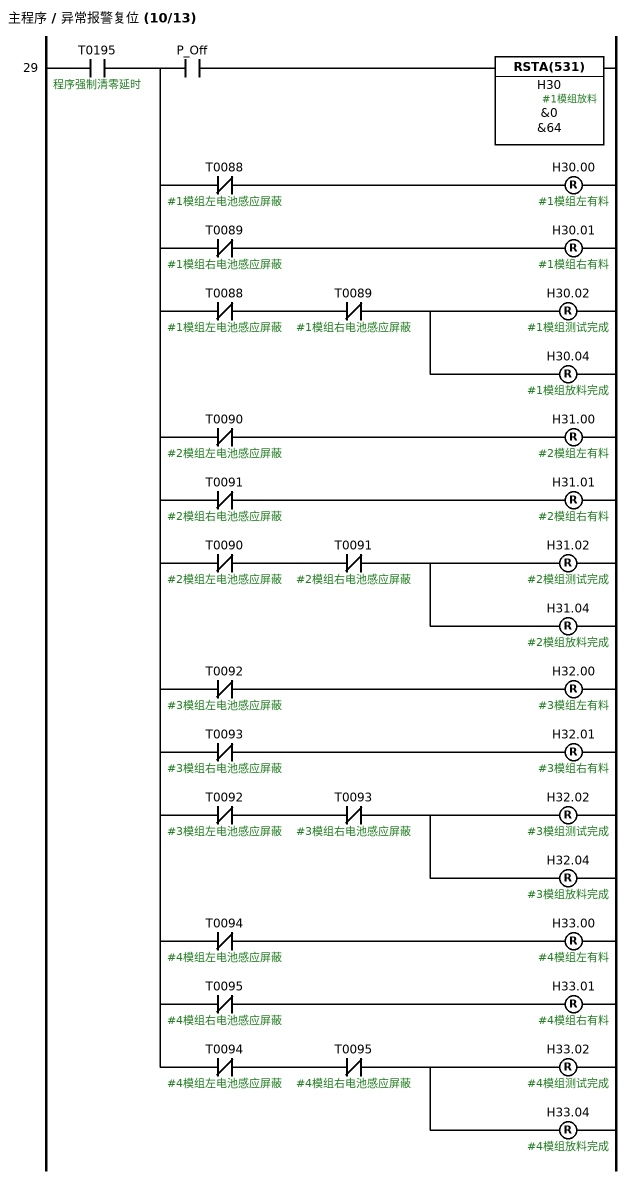
; [picture p17: 主程序 / 异常报警复位, rungs 29-29]
; rung 29
LD T0195  ; 程序强制清零延时
OUT TR0
AND P_Off
RSTA(531) H30 &0 &64  ; #1模组放料
LD TR0
ANDNOT T0088  ; #1模组左电池感应屏蔽
RSET H30.00  ; #1模组左有料
LD TR0
ANDNOT T0089  ; #1模组右电池感应屏蔽
RSET H30.01  ; #1模组右有料
LD TR0
ANDNOT T0088  ; #1模组左电池感应屏蔽
ANDNOT T0089  ; #1模组右电池感应屏蔽
RSET H30.02  ; #1模组测试完成
RSET H30.04  ; #1模组放料完成
LD TR0
ANDNOT T0090  ; #2模组左电池感应屏蔽
RSET H31.00  ; #2模组左有料
LD TR0
ANDNOT T0091  ; #2模组右电池感应屏蔽
RSET H31.01  ; #2模组右有料
LD TR0
ANDNOT T0090  ; #2模组左电池感应屏蔽
ANDNOT T0091  ; #2模组右电池感应屏蔽
RSET H31.02  ; #2模组测试完成
RSET H31.04  ; #2模组放料完成
LD TR0
ANDNOT T0092  ; #3模组左电池感应屏蔽
RSET H32.00  ; #3模组左有料
LD TR0
ANDNOT T0093  ; #3模组右电池感应屏蔽
RSET H32.01  ; #3模组右有料
LD TR0
ANDNOT T0092  ; #3模组左电池感应屏蔽
ANDNOT T0093  ; #3模组右电池感应屏蔽
RSET H32.02  ; #3模组测试完成
RSET H32.04  ; #3模组放料完成
LD TR0
ANDNOT T0094  ; #4模组左电池感应屏蔽
RSET H33.00  ; #4模组左有料
LD TR0
ANDNOT T0095  ; #4模组右电池感应屏蔽
RSET H33.01  ; #4模组右有料
LD TR0
ANDNOT T0094  ; #4模组左电池感应屏蔽
ANDNOT T0095  ; #4模组右电池感应屏蔽
RSET H33.02  ; #4模组测试完成
RSET H33.04  ; #4模组放料完成

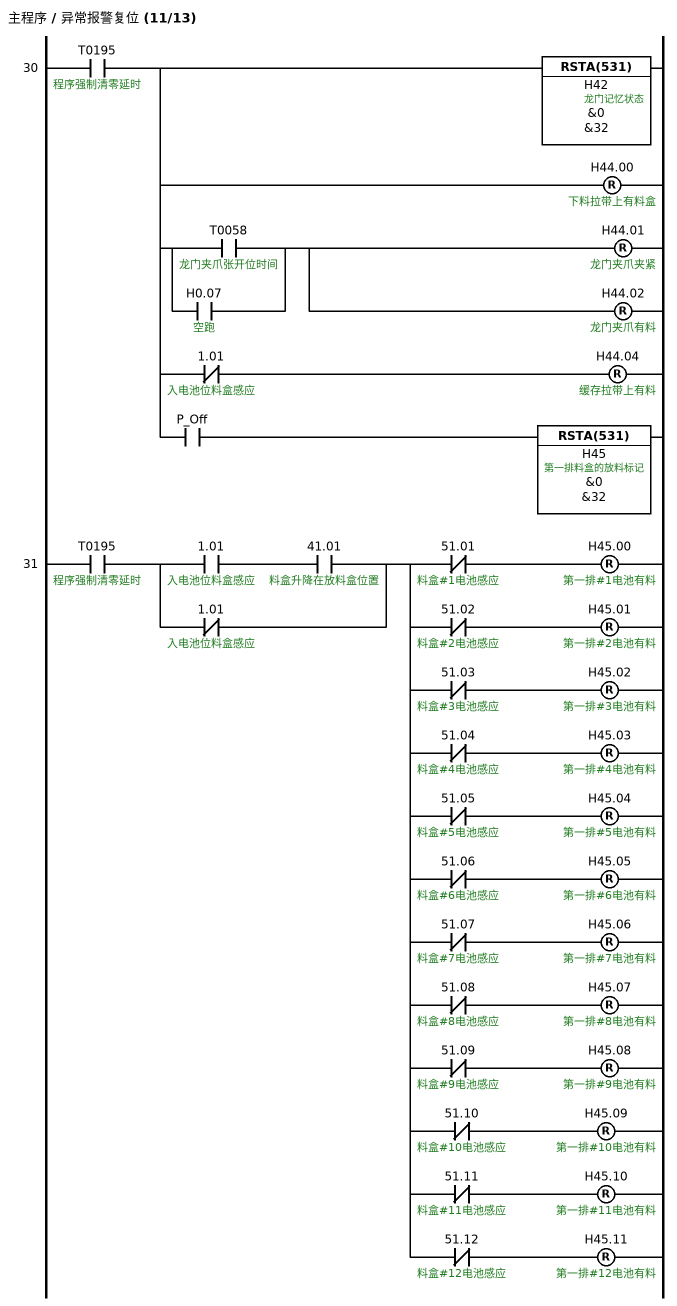
; rung 30
LD T0195  ; 程序强制清零延时
OUT TR0
RSTA(531) H42 &0 &32  ; 龙门记忆状态
RSET H44.00  ; 下料拉带上有料盒
LD T0058  ; 龙门夹爪张开位时间
OR H0.07  ; 空跑
ANDLD
RSET H44.01  ; 龙门夹爪夹紧
RSET H44.02  ; 龙门夹爪有料
LD TR0
ANDNOT 1.01  ; 入电池位料盒感应
RSET H44.04  ; 缓存拉带上有料
LD TR0
AND P_Off
RSTA(531) H45 &0 &32  ; 第一排料盒的放料标记
; rung 31
LD T0195  ; 程序强制清零延时
LD 1.01  ; 入电池位料盒感应
AND 41.01  ; 料盒升降在放料盒位置
ORNOT 1.01  ; 入电池位料盒感应
ANDLD
OUT TR0
ANDNOT 51.01  ; 料盒#1电池感应
RSET H45.00  ; 第一排#1电池有料
LD TR0
ANDNOT 51.02  ; 料盒#2电池感应
RSET H45.01  ; 第一排#2电池有料
LD TR0
ANDNOT 51.03  ; 料盒#3电池感应
RSET H45.02  ; 第一排#3电池有料
LD TR0
ANDNOT 51.04  ; 料盒#4电池感应
RSET H45.03  ; 第一排#4电池有料
LD TR0
ANDNOT 51.05  ; 料盒#5电池感应
RSET H45.04  ; 第一排#5电池有料
LD TR0
ANDNOT 51.06  ; 料盒#6电池感应
RSET H45.05  ; 第一排#6电池有料
LD TR0
ANDNOT 51.07  ; 料盒#7电池感应
RSET H45.06  ; 第一排#7电池有料
LD TR0
ANDNOT 51.08  ; 料盒#8电池感应
RSET H45.07  ; 第一排#8电池有料
LD TR0
ANDNOT 51.09  ; 料盒#9电池感应
RSET H45.08  ; 第一排#9电池有料
LD TR0
ANDNOT 51.10  ; 料盒#10电池感应
RSET H45.09  ; 第一排#10电池有料
LD TR0
ANDNOT 51.11  ; 料盒#11电池感应
RSET H45.10  ; 第一排#11电池有料
LD TR0
ANDNOT 51.12  ; 料盒#12电池感应
RSET H45.11  ; 第一排#12电池有料

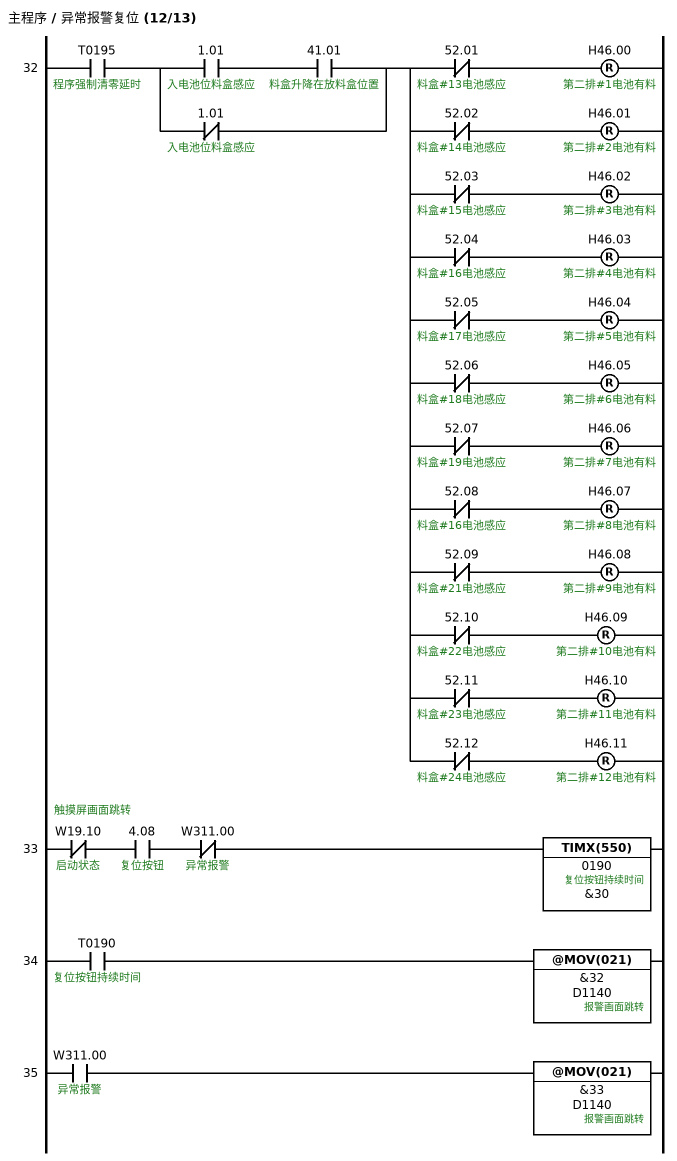
; rung 32
LD T0195  ; 程序强制清零延时
LD 1.01  ; 入电池位料盒感应
AND 41.01  ; 料盒升降在放料盒位置
ORNOT 1.01  ; 入电池位料盒感应
ANDLD
OUT TR0
ANDNOT 52.01  ; 料盒#13电池感应
RSET H46.00  ; 第二排#1电池有料
LD TR0
ANDNOT 52.02  ; 料盒#14电池感应
RSET H46.01  ; 第二排#2电池有料
LD TR0
ANDNOT 52.03  ; 料盒#15电池感应
RSET H46.02  ; 第二排#3电池有料
LD TR0
ANDNOT 52.04  ; 料盒#16电池感应
RSET H46.03  ; 第二排#4电池有料
LD TR0
ANDNOT 52.05  ; 料盒#17电池感应
RSET H46.04  ; 第二排#5电池有料
LD TR0
ANDNOT 52.06  ; 料盒#18电池感应
RSET H46.05  ; 第二排#6电池有料
LD TR0
ANDNOT 52.07  ; 料盒#19电池感应
RSET H46.06  ; 第二排#7电池有料
LD TR0
ANDNOT 52.08  ; 料盒#16电池感应
RSET H46.07  ; 第二排#8电池有料
LD TR0
ANDNOT 52.09  ; 料盒#21电池感应
RSET H46.08  ; 第二排#9电池有料
LD TR0
ANDNOT 52.10  ; 料盒#22电池感应
RSET H46.09  ; 第二排#10电池有料
LD TR0
ANDNOT 52.11  ; 料盒#23电池感应
RSET H46.10  ; 第二排#11电池有料
LD TR0
ANDNOT 52.12  ; 料盒#24电池感应
RSET H46.11  ; 第二排#12电池有料
; rung 33: 触摸屏画面跳转
LDNOT W19.10  ; 启动状态
AND 4.08  ; 复位按钮
ANDNOT W311.00  ; 异常报警
TIMX(550) 0190 &30  ; 复位按钮持续时间
; rung 34
LD T0190  ; 复位按钮持续时间
@MOV(021) &32 D1140  ; 报警画面跳转
; rung 35
LD W311.00  ; 异常报警
@MOV(021) &33 D1140  ; 报警画面跳转

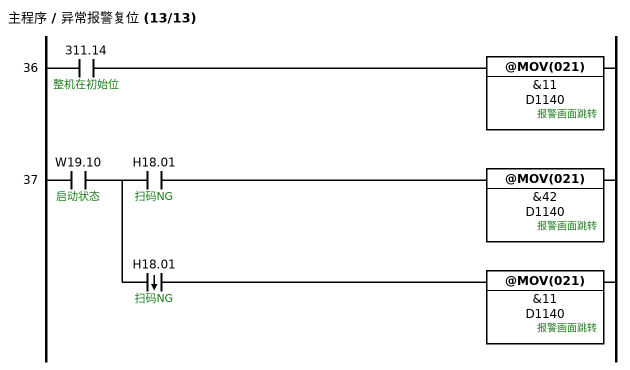
; rung 36
LD 311.14  ; 整机在初始位
@MOV(021) &11 D1140  ; 报警画面跳转
; rung 37
LD W19.10  ; 启动状态
OUT TR0
AND H18.01  ; 扫码NG
@MOV(021) &42 D1140  ; 报警画面跳转
LD TR0
%AND H18.01  ; 扫码NG
@MOV(021) &11 D1140  ; 报警画面跳转

### Section END
; rung 0
END(001)

## Program 传感器 (cyclic task 1)

### Section 感应器屏蔽

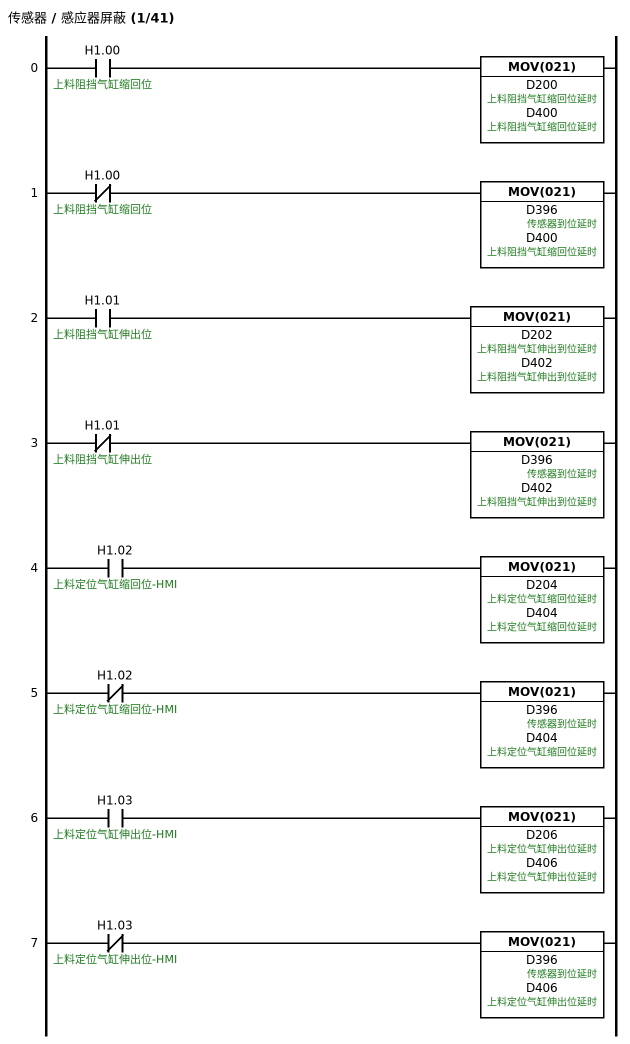
; rung 0
LD H1.00  ; 上料阻挡气缸缩回位
MOV(021) D200 D400  ; 上料阻挡气缸缩回位延时
; rung 1
LDNOT H1.00  ; 上料阻挡气缸缩回位
MOV(021) D396 D400  ; 传感器到位延时, 上料阻挡气缸缩回位延时
; rung 2
LD H1.01  ; 上料阻挡气缸伸出位
MOV(021) D202 D402  ; 上料阻挡气缸伸出到位延时
; rung 3
LDNOT H1.01  ; 上料阻挡气缸伸出位
MOV(021) D396 D402  ; 传感器到位延时, 上料阻挡气缸伸出到位延时
; rung 4
LD H1.02  ; 上料定位气缸缩回位-HMI
MOV(021) D204 D404  ; 上料定位气缸缩回位延时
; rung 5
LDNOT H1.02  ; 上料定位气缸缩回位-HMI
MOV(021) D396 D404  ; 传感器到位延时, 上料定位气缸缩回位延时
; rung 6
LD H1.03  ; 上料定位气缸伸出位-HMI
MOV(021) D206 D406  ; 上料定位气缸伸出位延时
; rung 7
LDNOT H1.03  ; 上料定位气缸伸出位-HMI
MOV(021) D396 D406  ; 传感器到位延时, 上料定位气缸伸出位延时

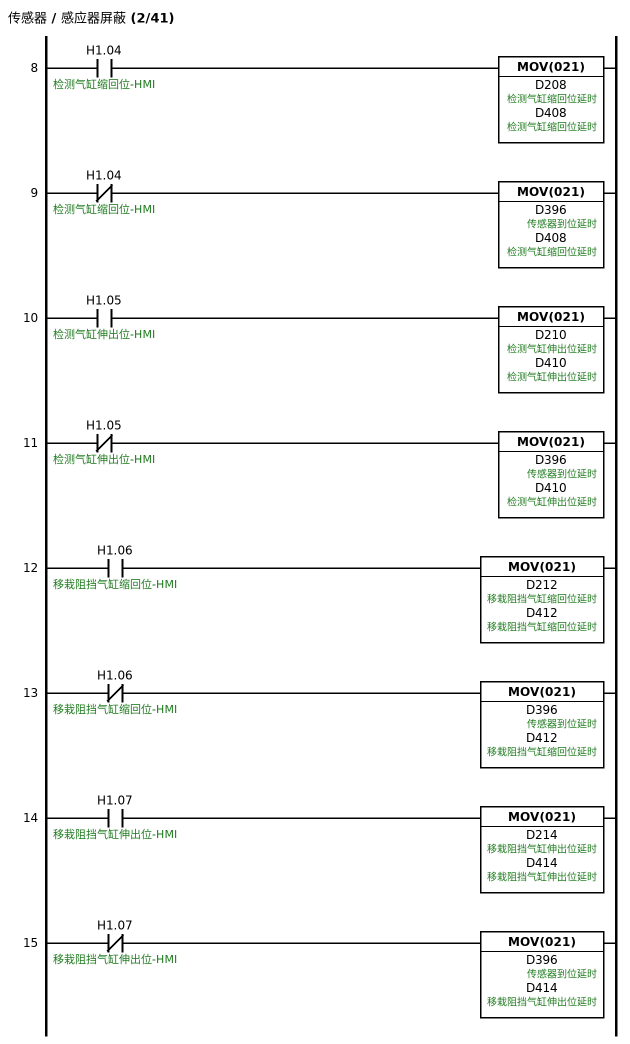
; rung 8
LD H1.04  ; 检测气缸缩回位-HMI
MOV(021) D208 D408  ; 检测气缸缩回位延时
; rung 9
LDNOT H1.04  ; 检测气缸缩回位-HMI
MOV(021) D396 D408  ; 传感器到位延时, 检测气缸缩回位延时
; rung 10
LD H1.05  ; 检测气缸伸出位-HMI
MOV(021) D210 D410  ; 检测气缸伸出位延时
; rung 11
LDNOT H1.05  ; 检测气缸伸出位-HMI
MOV(021) D396 D410  ; 传感器到位延时, 检测气缸伸出位延时
; rung 12
LD H1.06  ; 移栽阻挡气缸缩回位-HMI
MOV(021) D212 D412  ; 移栽阻挡气缸缩回位延时
; rung 13
LDNOT H1.06  ; 移栽阻挡气缸缩回位-HMI
MOV(021) D396 D412  ; 传感器到位延时, 移栽阻挡气缸缩回位延时
; rung 14
LD H1.07  ; 移栽阻挡气缸伸出位-HMI
MOV(021) D214 D414  ; 移栽阻挡气缸伸出位延时
; rung 15
LDNOT H1.07  ; 移栽阻挡气缸伸出位-HMI
MOV(021) D396 D414  ; 传感器到位延时, 移栽阻挡气缸伸出位延时

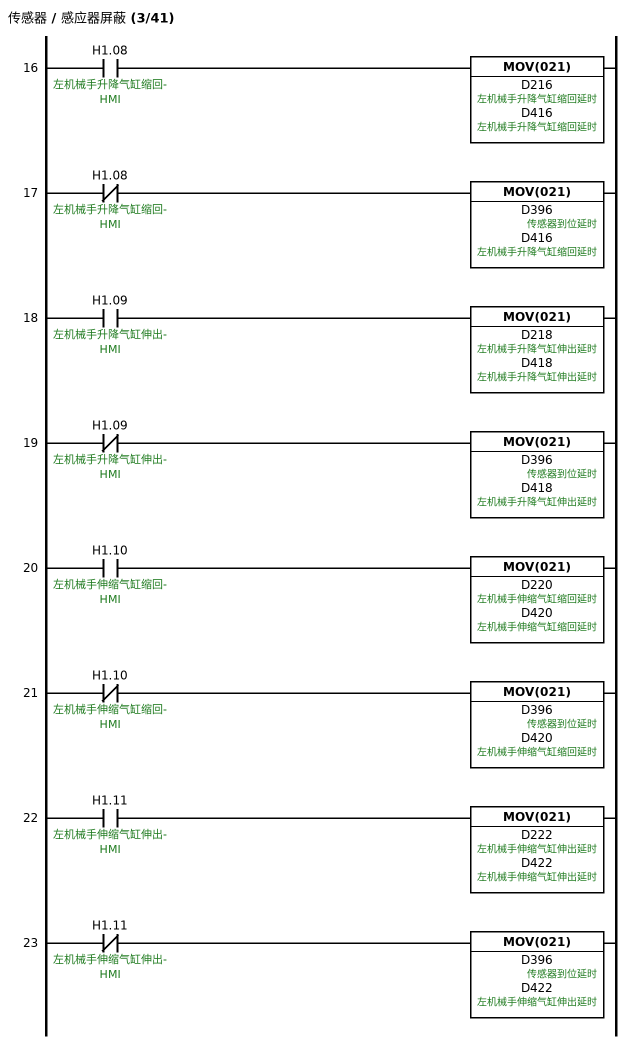
; rung 16
LD H1.08  ; 左机械手升降气缸缩回-HMI
MOV(021) D216 D416  ; 左机械手升降气缸缩回延时
; rung 17
LDNOT H1.08  ; 左机械手升降气缸缩回-HMI
MOV(021) D396 D416  ; 传感器到位延时, 左机械手升降气缸缩回延时
; rung 18
LD H1.09  ; 左机械手升降气缸伸出-HMI
MOV(021) D218 D418  ; 左机械手升降气缸伸出延时
; rung 19
LDNOT H1.09  ; 左机械手升降气缸伸出-HMI
MOV(021) D396 D418  ; 传感器到位延时, 左机械手升降气缸伸出延时
; rung 20
LD H1.10  ; 左机械手伸缩气缸缩回-HMI
MOV(021) D220 D420  ; 左机械手伸缩气缸缩回延时
; rung 21
LDNOT H1.10  ; 左机械手伸缩气缸缩回-HMI
MOV(021) D396 D420  ; 传感器到位延时, 左机械手伸缩气缸缩回延时
; rung 22
LD H1.11  ; 左机械手伸缩气缸伸出-HMI
MOV(021) D222 D422  ; 左机械手伸缩气缸伸出延时
; rung 23
LDNOT H1.11  ; 左机械手伸缩气缸伸出-HMI
MOV(021) D396 D422  ; 传感器到位延时, 左机械手伸缩气缸伸出延时

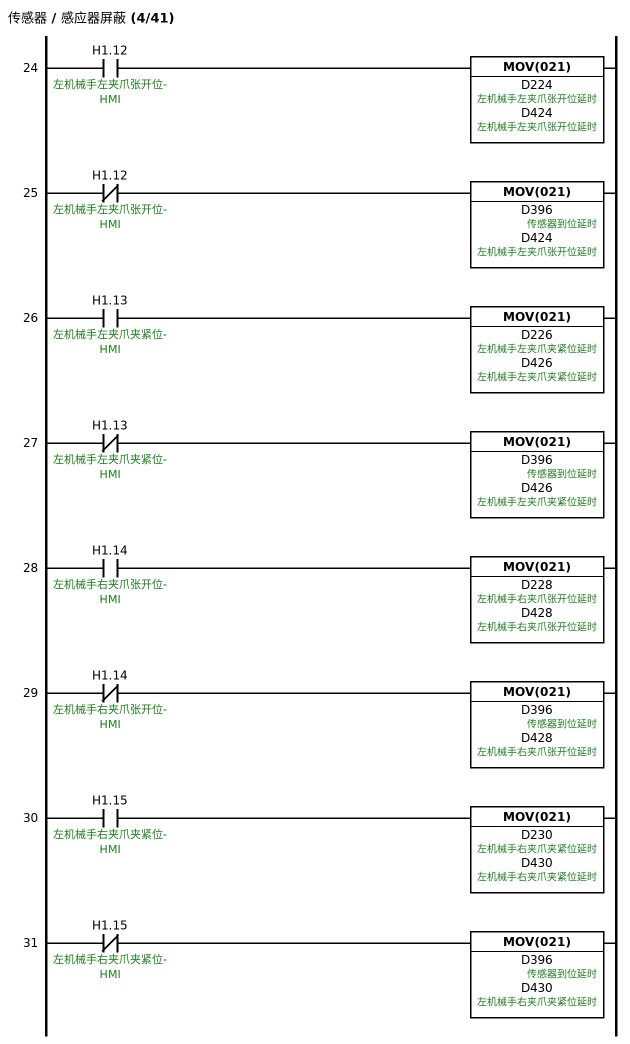
; rung 24
LD H1.12  ; 左机械手左夹爪张开位-HMI
MOV(021) D224 D424  ; 左机械手左夹爪张开位延时
; rung 25
LDNOT H1.12  ; 左机械手左夹爪张开位-HMI
MOV(021) D396 D424  ; 传感器到位延时, 左机械手左夹爪张开位延时
; rung 26
LD H1.13  ; 左机械手左夹爪夹紧位-HMI
MOV(021) D226 D426  ; 左机械手左夹爪夹紧位延时
; rung 27
LDNOT H1.13  ; 左机械手左夹爪夹紧位-HMI
MOV(021) D396 D426  ; 传感器到位延时, 左机械手左夹爪夹紧位延时
; rung 28
LD H1.14  ; 左机械手右夹爪张开位-HMI
MOV(021) D228 D428  ; 左机械手右夹爪张开位延时
; rung 29
LDNOT H1.14  ; 左机械手右夹爪张开位-HMI
MOV(021) D396 D428  ; 传感器到位延时, 左机械手右夹爪张开位延时
; rung 30
LD H1.15  ; 左机械手右夹爪夹紧位-HMI
MOV(021) D230 D430  ; 左机械手右夹爪夹紧位延时
; rung 31
LDNOT H1.15  ; 左机械手右夹爪夹紧位-HMI
MOV(021) D396 D430  ; 传感器到位延时, 左机械手右夹爪夹紧位延时

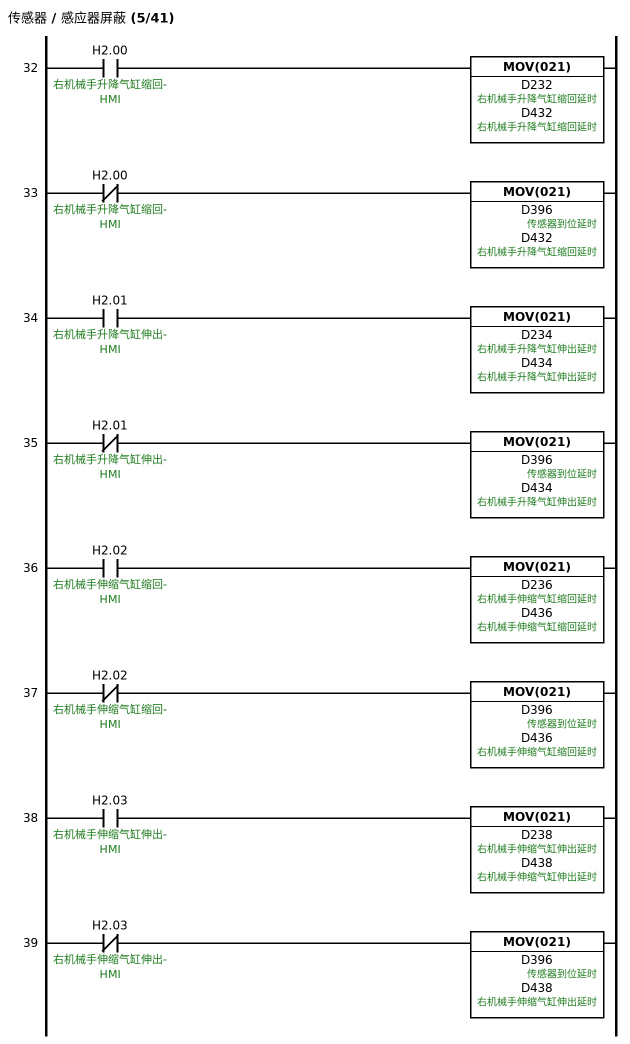
; rung 32
LD H2.00  ; 右机械手升降气缸缩回-HMI
MOV(021) D232 D432  ; 右机械手升降气缸缩回延时
; rung 33
LDNOT H2.00  ; 右机械手升降气缸缩回-HMI
MOV(021) D396 D432  ; 传感器到位延时, 右机械手升降气缸缩回延时
; rung 34
LD H2.01  ; 右机械手升降气缸伸出-HMI
MOV(021) D234 D434  ; 右机械手升降气缸伸出延时
; rung 35
LDNOT H2.01  ; 右机械手升降气缸伸出-HMI
MOV(021) D396 D434  ; 传感器到位延时, 右机械手升降气缸伸出延时
; rung 36
LD H2.02  ; 右机械手伸缩气缸缩回-HMI
MOV(021) D236 D436  ; 右机械手伸缩气缸缩回延时
; rung 37
LDNOT H2.02  ; 右机械手伸缩气缸缩回-HMI
MOV(021) D396 D436  ; 传感器到位延时, 右机械手伸缩气缸缩回延时
; rung 38
LD H2.03  ; 右机械手伸缩气缸伸出-HMI
MOV(021) D238 D438  ; 右机械手伸缩气缸伸出延时
; rung 39
LDNOT H2.03  ; 右机械手伸缩气缸伸出-HMI
MOV(021) D396 D438  ; 传感器到位延时, 右机械手伸缩气缸伸出延时

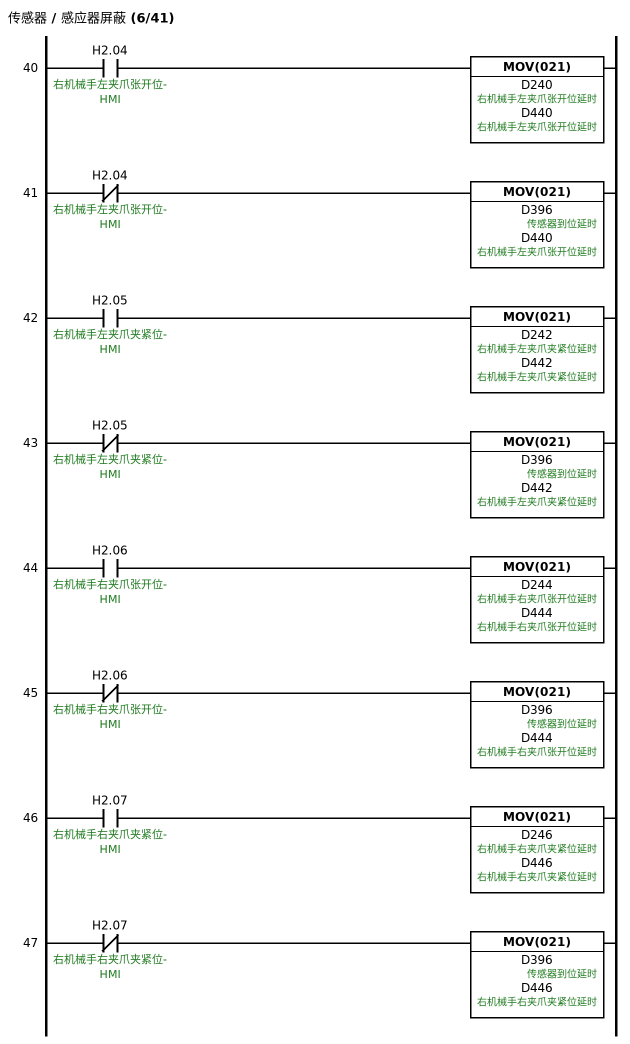
; rung 40
LD H2.04  ; 右机械手左夹爪张开位-HMI
MOV(021) D240 D440  ; 右机械手左夹爪张开位延时
; rung 41
LDNOT H2.04  ; 右机械手左夹爪张开位-HMI
MOV(021) D396 D440  ; 传感器到位延时, 右机械手左夹爪张开位延时
; rung 42
LD H2.05  ; 右机械手左夹爪夹紧位-HMI
MOV(021) D242 D442  ; 右机械手左夹爪夹紧位延时
; rung 43
LDNOT H2.05  ; 右机械手左夹爪夹紧位-HMI
MOV(021) D396 D442  ; 传感器到位延时, 右机械手左夹爪夹紧位延时
; rung 44
LD H2.06  ; 右机械手右夹爪张开位-HMI
MOV(021) D244 D444  ; 右机械手右夹爪张开位延时
; rung 45
LDNOT H2.06  ; 右机械手右夹爪张开位-HMI
MOV(021) D396 D444  ; 传感器到位延时, 右机械手右夹爪张开位延时
; rung 46
LD H2.07  ; 右机械手右夹爪夹紧位-HMI
MOV(021) D246 D446  ; 右机械手右夹爪夹紧位延时
; rung 47
LDNOT H2.07  ; 右机械手右夹爪夹紧位-HMI
MOV(021) D396 D446  ; 传感器到位延时, 右机械手右夹爪夹紧位延时

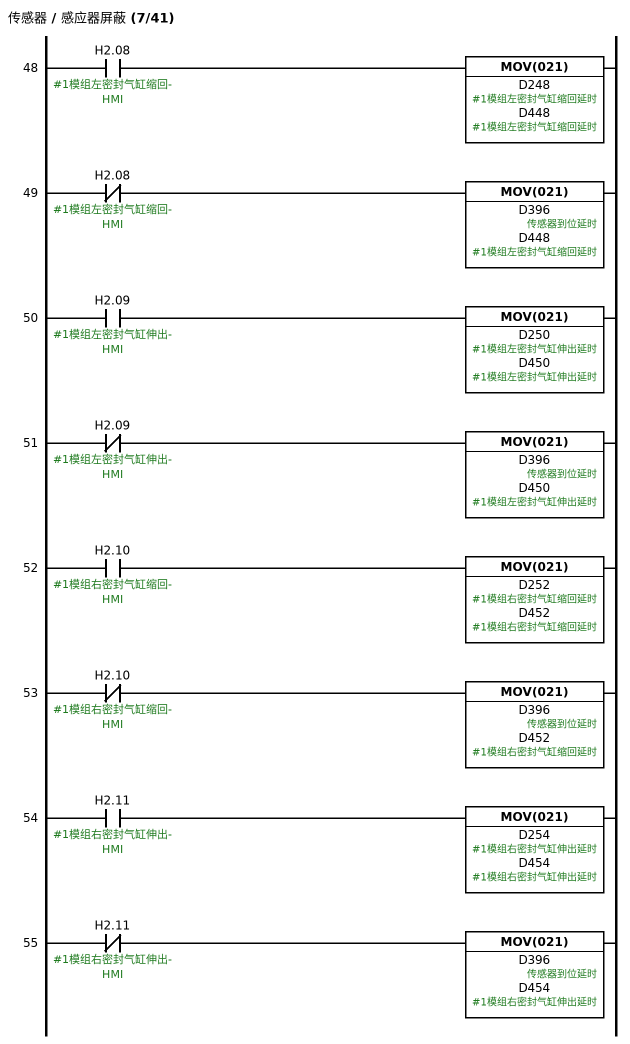
; rung 48
LD H2.08  ; #1模组左密封气缸缩回-HMI
MOV(021) D248 D448  ; #1模组左密封气缸缩回延时
; rung 49
LDNOT H2.08  ; #1模组左密封气缸缩回-HMI
MOV(021) D396 D448  ; 传感器到位延时, #1模组左密封气缸缩回延时
; rung 50
LD H2.09  ; #1模组左密封气缸伸出-HMI
MOV(021) D250 D450  ; #1模组左密封气缸伸出延时
; rung 51
LDNOT H2.09  ; #1模组左密封气缸伸出-HMI
MOV(021) D396 D450  ; 传感器到位延时, #1模组左密封气缸伸出延时
; rung 52
LD H2.10  ; #1模组右密封气缸缩回-HMI
MOV(021) D252 D452  ; #1模组右密封气缸缩回延时
; rung 53
LDNOT H2.10  ; #1模组右密封气缸缩回-HMI
MOV(021) D396 D452  ; 传感器到位延时, #1模组右密封气缸缩回延时
; rung 54
LD H2.11  ; #1模组右密封气缸伸出-HMI
MOV(021) D254 D454  ; #1模组右密封气缸伸出延时
; rung 55
LDNOT H2.11  ; #1模组右密封气缸伸出-HMI
MOV(021) D396 D454  ; 传感器到位延时, #1模组右密封气缸伸出延时

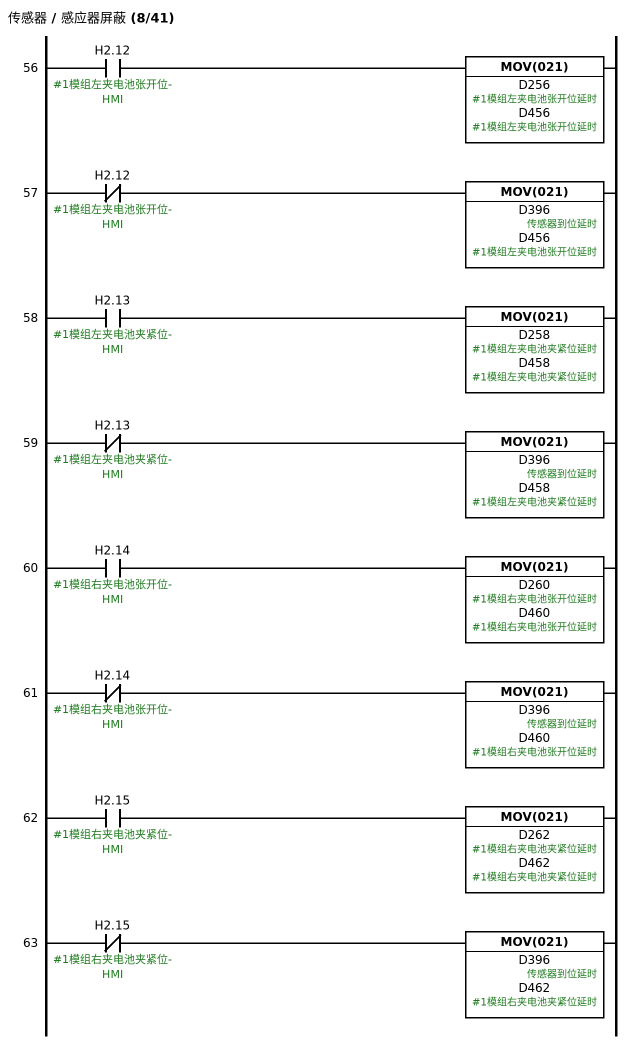
; rung 56
LD H2.12  ; #1模组左夹电池张开位-HMI
MOV(021) D256 D456  ; #1模组左夹电池张开位延时
; rung 57
LDNOT H2.12  ; #1模组左夹电池张开位-HMI
MOV(021) D396 D456  ; 传感器到位延时, #1模组左夹电池张开位延时
; rung 58
LD H2.13  ; #1模组左夹电池夹紧位-HMI
MOV(021) D258 D458  ; #1模组左夹电池夹紧位延时
; rung 59
LDNOT H2.13  ; #1模组左夹电池夹紧位-HMI
MOV(021) D396 D458  ; 传感器到位延时, #1模组左夹电池夹紧位延时
; rung 60
LD H2.14  ; #1模组右夹电池张开位-HMI
MOV(021) D260 D460  ; #1模组右夹电池张开位延时
; rung 61
LDNOT H2.14  ; #1模组右夹电池张开位-HMI
MOV(021) D396 D460  ; 传感器到位延时, #1模组右夹电池张开位延时
; rung 62
LD H2.15  ; #1模组右夹电池夹紧位-HMI
MOV(021) D262 D462  ; #1模组右夹电池夹紧位延时
; rung 63
LDNOT H2.15  ; #1模组右夹电池夹紧位-HMI
MOV(021) D396 D462  ; 传感器到位延时, #1模组右夹电池夹紧位延时

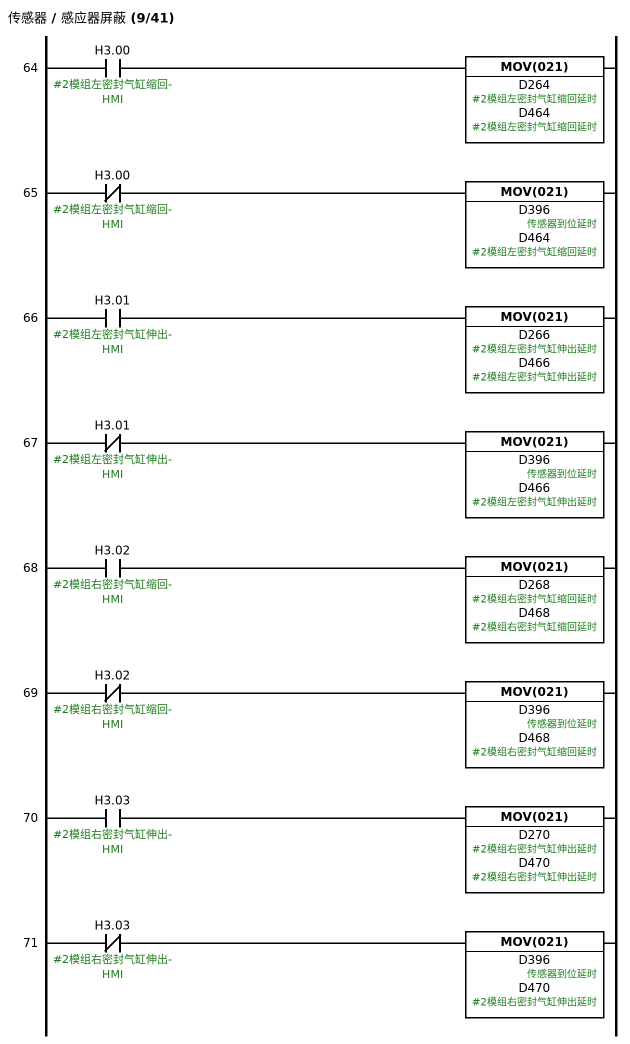
; rung 64
LD H3.00  ; #2模组左密封气缸缩回-HMI
MOV(021) D264 D464  ; #2模组左密封气缸缩回延时
; rung 65
LDNOT H3.00  ; #2模组左密封气缸缩回-HMI
MOV(021) D396 D464  ; 传感器到位延时, #2模组左密封气缸缩回延时
; rung 66
LD H3.01  ; #2模组左密封气缸伸出-HMI
MOV(021) D266 D466  ; #2模组左密封气缸伸出延时
; rung 67
LDNOT H3.01  ; #2模组左密封气缸伸出-HMI
MOV(021) D396 D466  ; 传感器到位延时, #2模组左密封气缸伸出延时
; rung 68
LD H3.02  ; #2模组右密封气缸缩回-HMI
MOV(021) D268 D468  ; #2模组右密封气缸缩回延时
; rung 69
LDNOT H3.02  ; #2模组右密封气缸缩回-HMI
MOV(021) D396 D468  ; 传感器到位延时, #2模组右密封气缸缩回延时
; rung 70
LD H3.03  ; #2模组右密封气缸伸出-HMI
MOV(021) D270 D470  ; #2模组右密封气缸伸出延时
; rung 71
LDNOT H3.03  ; #2模组右密封气缸伸出-HMI
MOV(021) D396 D470  ; 传感器到位延时, #2模组右密封气缸伸出延时

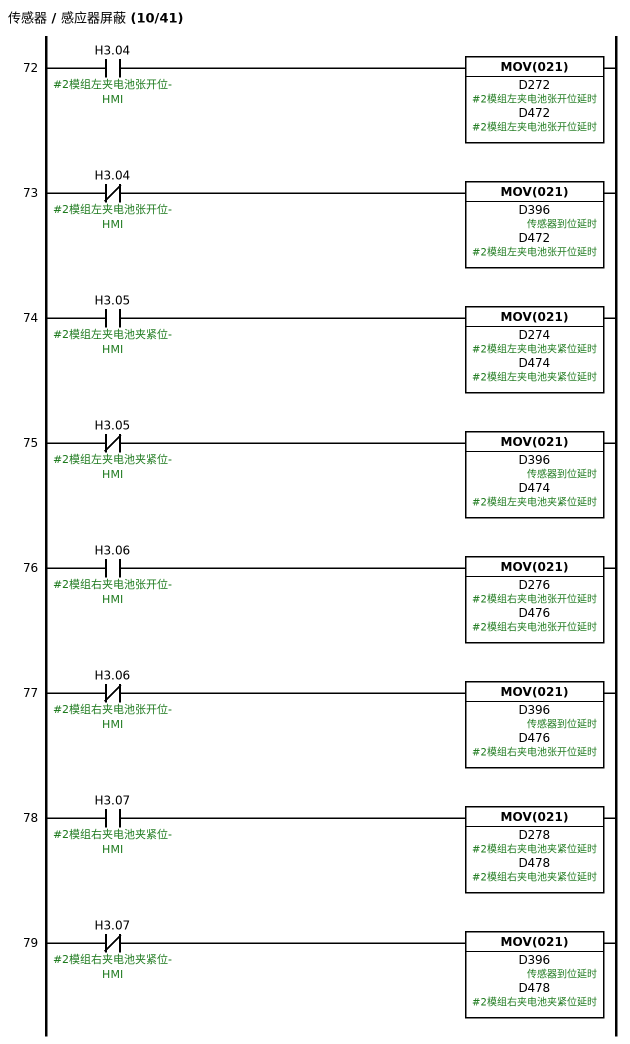
; rung 72
LD H3.04  ; #2模组左夹电池张开位-HMI
MOV(021) D272 D472  ; #2模组左夹电池张开位延时
; rung 73
LDNOT H3.04  ; #2模组左夹电池张开位-HMI
MOV(021) D396 D472  ; 传感器到位延时, #2模组左夹电池张开位延时
; rung 74
LD H3.05  ; #2模组左夹电池夹紧位-HMI
MOV(021) D274 D474  ; #2模组左夹电池夹紧位延时
; rung 75
LDNOT H3.05  ; #2模组左夹电池夹紧位-HMI
MOV(021) D396 D474  ; 传感器到位延时, #2模组左夹电池夹紧位延时
; rung 76
LD H3.06  ; #2模组右夹电池张开位-HMI
MOV(021) D276 D476  ; #2模组右夹电池张开位延时
; rung 77
LDNOT H3.06  ; #2模组右夹电池张开位-HMI
MOV(021) D396 D476  ; 传感器到位延时, #2模组右夹电池张开位延时
; rung 78
LD H3.07  ; #2模组右夹电池夹紧位-HMI
MOV(021) D278 D478  ; #2模组右夹电池夹紧位延时
; rung 79
LDNOT H3.07  ; #2模组右夹电池夹紧位-HMI
MOV(021) D396 D478  ; 传感器到位延时, #2模组右夹电池夹紧位延时

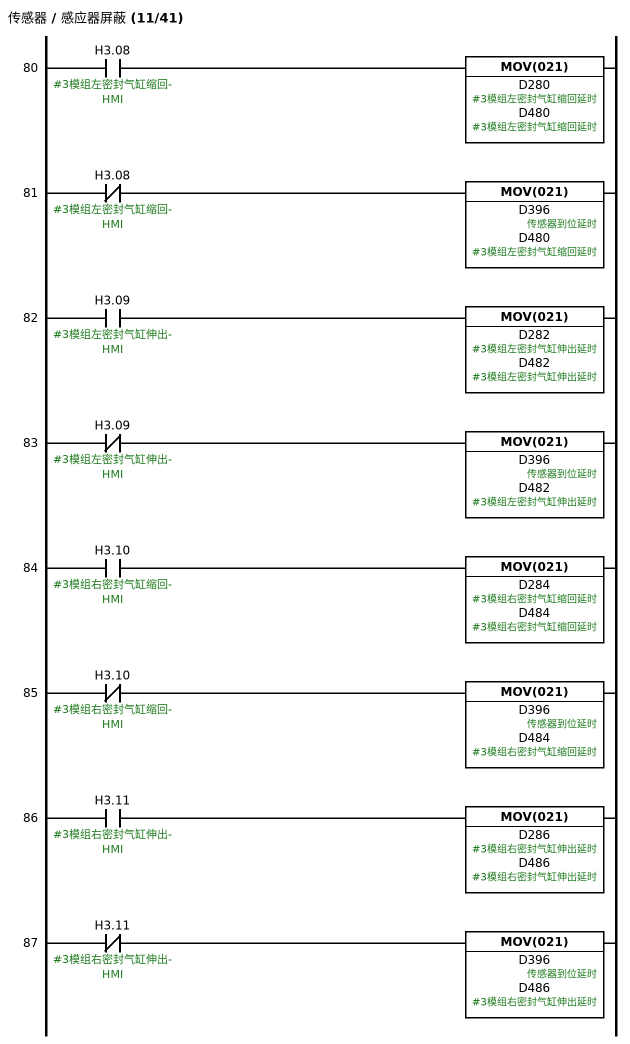
; rung 80
LD H3.08  ; #3模组左密封气缸缩回-HMI
MOV(021) D280 D480  ; #3模组左密封气缸缩回延时
; rung 81
LDNOT H3.08  ; #3模组左密封气缸缩回-HMI
MOV(021) D396 D480  ; 传感器到位延时, #3模组左密封气缸缩回延时
; rung 82
LD H3.09  ; #3模组左密封气缸伸出-HMI
MOV(021) D282 D482  ; #3模组左密封气缸伸出延时
; rung 83
LDNOT H3.09  ; #3模组左密封气缸伸出-HMI
MOV(021) D396 D482  ; 传感器到位延时, #3模组左密封气缸伸出延时
; rung 84
LD H3.10  ; #3模组右密封气缸缩回-HMI
MOV(021) D284 D484  ; #3模组右密封气缸缩回延时
; rung 85
LDNOT H3.10  ; #3模组右密封气缸缩回-HMI
MOV(021) D396 D484  ; 传感器到位延时, #3模组右密封气缸缩回延时
; rung 86
LD H3.11  ; #3模组右密封气缸伸出-HMI
MOV(021) D286 D486  ; #3模组右密封气缸伸出延时
; rung 87
LDNOT H3.11  ; #3模组右密封气缸伸出-HMI
MOV(021) D396 D486  ; 传感器到位延时, #3模组右密封气缸伸出延时

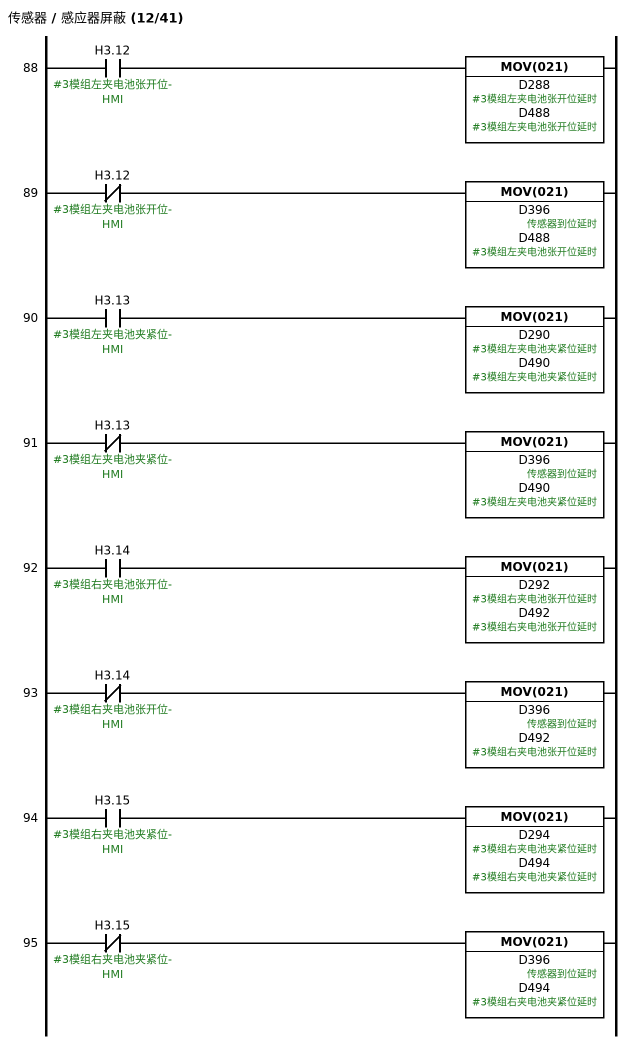
; rung 88
LD H3.12  ; #3模组左夹电池张开位-HMI
MOV(021) D288 D488  ; #3模组左夹电池张开位延时
; rung 89
LDNOT H3.12  ; #3模组左夹电池张开位-HMI
MOV(021) D396 D488  ; 传感器到位延时, #3模组左夹电池张开位延时
; rung 90
LD H3.13  ; #3模组左夹电池夹紧位-HMI
MOV(021) D290 D490  ; #3模组左夹电池夹紧位延时
; rung 91
LDNOT H3.13  ; #3模组左夹电池夹紧位-HMI
MOV(021) D396 D490  ; 传感器到位延时, #3模组左夹电池夹紧位延时
; rung 92
LD H3.14  ; #3模组右夹电池张开位-HMI
MOV(021) D292 D492  ; #3模组右夹电池张开位延时
; rung 93
LDNOT H3.14  ; #3模组右夹电池张开位-HMI
MOV(021) D396 D492  ; 传感器到位延时, #3模组右夹电池张开位延时
; rung 94
LD H3.15  ; #3模组右夹电池夹紧位-HMI
MOV(021) D294 D494  ; #3模组右夹电池夹紧位延时
; rung 95
LDNOT H3.15  ; #3模组右夹电池夹紧位-HMI
MOV(021) D396 D494  ; 传感器到位延时, #3模组右夹电池夹紧位延时

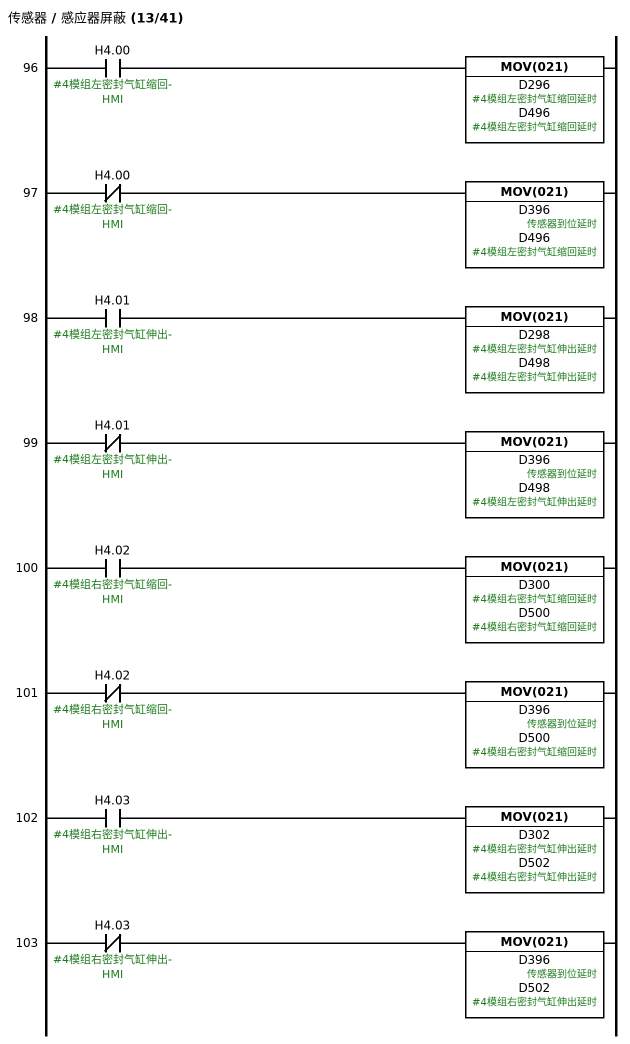
; rung 96
LD H4.00  ; #4模组左密封气缸缩回-HMI
MOV(021) D296 D496  ; #4模组左密封气缸缩回延时
; rung 97
LDNOT H4.00  ; #4模组左密封气缸缩回-HMI
MOV(021) D396 D496  ; 传感器到位延时, #4模组左密封气缸缩回延时
; rung 98
LD H4.01  ; #4模组左密封气缸伸出-HMI
MOV(021) D298 D498  ; #4模组左密封气缸伸出延时
; rung 99
LDNOT H4.01  ; #4模组左密封气缸伸出-HMI
MOV(021) D396 D498  ; 传感器到位延时, #4模组左密封气缸伸出延时
; rung 100
LD H4.02  ; #4模组右密封气缸缩回-HMI
MOV(021) D300 D500  ; #4模组右密封气缸缩回延时
; rung 101
LDNOT H4.02  ; #4模组右密封气缸缩回-HMI
MOV(021) D396 D500  ; 传感器到位延时, #4模组右密封气缸缩回延时
; rung 102
LD H4.03  ; #4模组右密封气缸伸出-HMI
MOV(021) D302 D502  ; #4模组右密封气缸伸出延时
; rung 103
LDNOT H4.03  ; #4模组右密封气缸伸出-HMI
MOV(021) D396 D502  ; 传感器到位延时, #4模组右密封气缸伸出延时

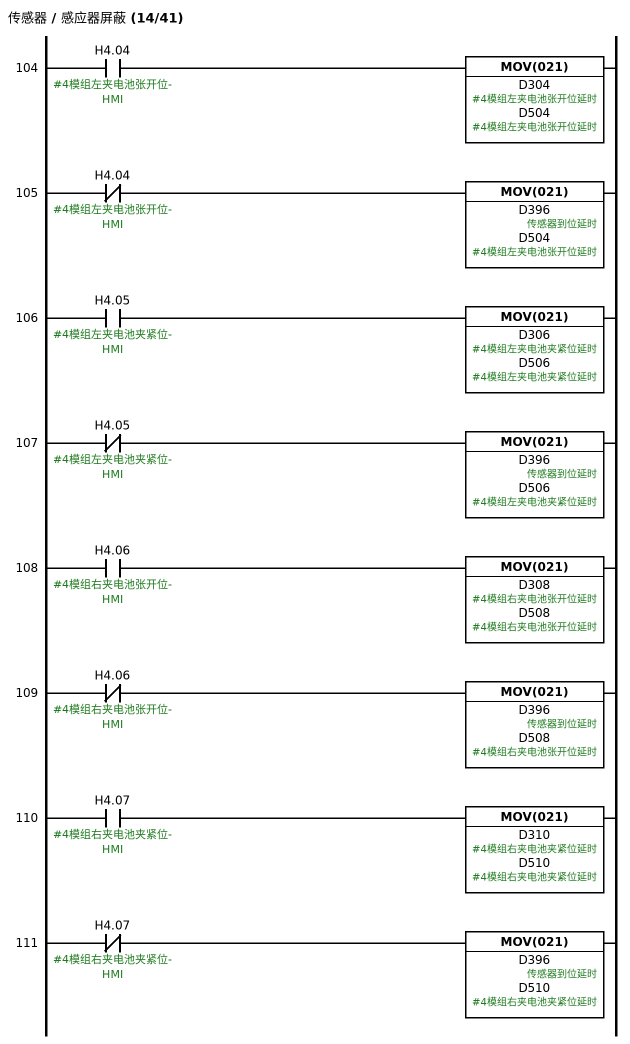
; rung 104
LD H4.04  ; #4模组左夹电池张开位-HMI
MOV(021) D304 D504  ; #4模组左夹电池张开位延时
; rung 105
LDNOT H4.04  ; #4模组左夹电池张开位-HMI
MOV(021) D396 D504  ; 传感器到位延时, #4模组左夹电池张开位延时
; rung 106
LD H4.05  ; #4模组左夹电池夹紧位-HMI
MOV(021) D306 D506  ; #4模组左夹电池夹紧位延时
; rung 107
LDNOT H4.05  ; #4模组左夹电池夹紧位-HMI
MOV(021) D396 D506  ; 传感器到位延时, #4模组左夹电池夹紧位延时
; rung 108
LD H4.06  ; #4模组右夹电池张开位-HMI
MOV(021) D308 D508  ; #4模组右夹电池张开位延时
; rung 109
LDNOT H4.06  ; #4模组右夹电池张开位-HMI
MOV(021) D396 D508  ; 传感器到位延时, #4模组右夹电池张开位延时
; rung 110
LD H4.07  ; #4模组右夹电池夹紧位-HMI
MOV(021) D310 D510  ; #4模组右夹电池夹紧位延时
; rung 111
LDNOT H4.07  ; #4模组右夹电池夹紧位-HMI
MOV(021) D396 D510  ; 传感器到位延时, #4模组右夹电池夹紧位延时

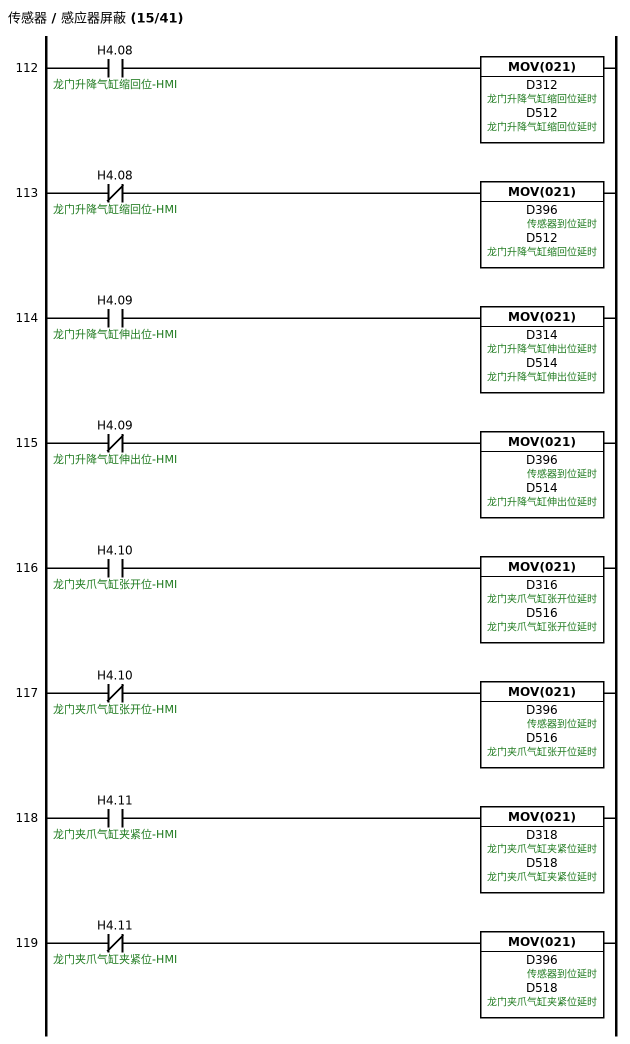
; rung 112
LD H4.08  ; 龙门升降气缸缩回位-HMI
MOV(021) D312 D512  ; 龙门升降气缸缩回位延时
; rung 113
LDNOT H4.08  ; 龙门升降气缸缩回位-HMI
MOV(021) D396 D512  ; 传感器到位延时, 龙门升降气缸缩回位延时
; rung 114
LD H4.09  ; 龙门升降气缸伸出位-HMI
MOV(021) D314 D514  ; 龙门升降气缸伸出位延时
; rung 115
LDNOT H4.09  ; 龙门升降气缸伸出位-HMI
MOV(021) D396 D514  ; 传感器到位延时, 龙门升降气缸伸出位延时
; rung 116
LD H4.10  ; 龙门夹爪气缸张开位-HMI
MOV(021) D316 D516  ; 龙门夹爪气缸张开位延时
; rung 117
LDNOT H4.10  ; 龙门夹爪气缸张开位-HMI
MOV(021) D396 D516  ; 传感器到位延时, 龙门夹爪气缸张开位延时
; rung 118
LD H4.11  ; 龙门夹爪气缸夹紧位-HMI
MOV(021) D318 D518  ; 龙门夹爪气缸夹紧位延时
; rung 119
LDNOT H4.11  ; 龙门夹爪气缸夹紧位-HMI
MOV(021) D396 D518  ; 传感器到位延时, 龙门夹爪气缸夹紧位延时

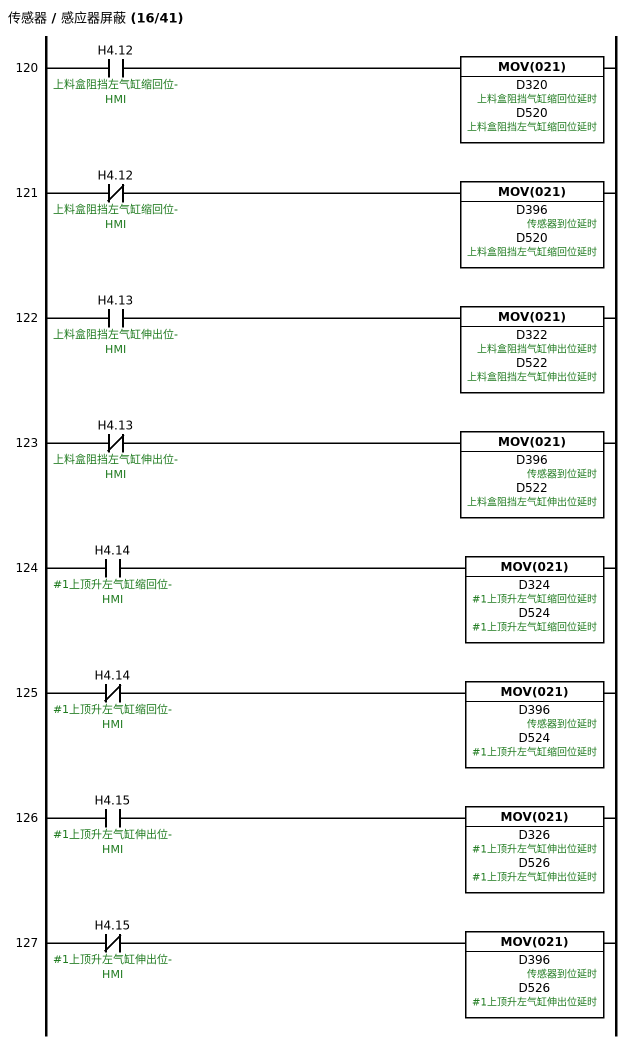
; rung 120
LD H4.12  ; 上料盒阻挡左气缸缩回位-HMI
MOV(021) D320 D520  ; 上料盒阻挡气缸缩回位延时, 上料盒阻挡左气缸缩回位延时
; rung 121
LDNOT H4.12  ; 上料盒阻挡左气缸缩回位-HMI
MOV(021) D396 D520  ; 传感器到位延时, 上料盒阻挡左气缸缩回位延时
; rung 122
LD H4.13  ; 上料盒阻挡左气缸伸出位-HMI
MOV(021) D322 D522  ; 上料盒阻挡气缸伸出位延时, 上料盒阻挡左气缸伸出位延时
; rung 123
LDNOT H4.13  ; 上料盒阻挡左气缸伸出位-HMI
MOV(021) D396 D522  ; 传感器到位延时, 上料盒阻挡左气缸伸出位延时
; rung 124
LD H4.14  ; #1上顶升左气缸缩回位-HMI
MOV(021) D324 D524  ; #1上顶升左气缸缩回位延时
; rung 125
LDNOT H4.14  ; #1上顶升左气缸缩回位-HMI
MOV(021) D396 D524  ; 传感器到位延时, #1上顶升左气缸缩回位延时
; rung 126
LD H4.15  ; #1上顶升左气缸伸出位-HMI
MOV(021) D326 D526  ; #1上顶升左气缸伸出位延时
; rung 127
LDNOT H4.15  ; #1上顶升左气缸伸出位-HMI
MOV(021) D396 D526  ; 传感器到位延时, #1上顶升左气缸伸出位延时

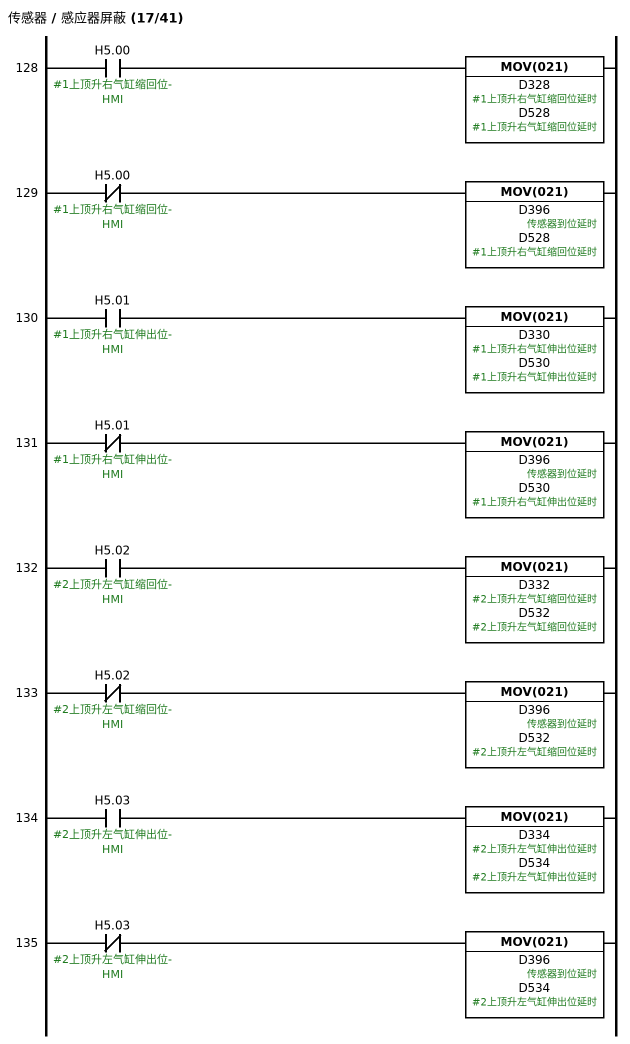
; rung 128
LD H5.00  ; #1上顶升右气缸缩回位-HMI
MOV(021) D328 D528  ; #1上顶升右气缸缩回位延时
; rung 129
LDNOT H5.00  ; #1上顶升右气缸缩回位-HMI
MOV(021) D396 D528  ; 传感器到位延时, #1上顶升右气缸缩回位延时
; rung 130
LD H5.01  ; #1上顶升右气缸伸出位-HMI
MOV(021) D330 D530  ; #1上顶升右气缸伸出位延时
; rung 131
LDNOT H5.01  ; #1上顶升右气缸伸出位-HMI
MOV(021) D396 D530  ; 传感器到位延时, #1上顶升右气缸伸出位延时
; rung 132
LD H5.02  ; #2上顶升左气缸缩回位-HMI
MOV(021) D332 D532  ; #2上顶升左气缸缩回位延时
; rung 133
LDNOT H5.02  ; #2上顶升左气缸缩回位-HMI
MOV(021) D396 D532  ; 传感器到位延时, #2上顶升左气缸缩回位延时
; rung 134
LD H5.03  ; #2上顶升左气缸伸出位-HMI
MOV(021) D334 D534  ; #2上顶升左气缸伸出位延时
; rung 135
LDNOT H5.03  ; #2上顶升左气缸伸出位-HMI
MOV(021) D396 D534  ; 传感器到位延时, #2上顶升左气缸伸出位延时

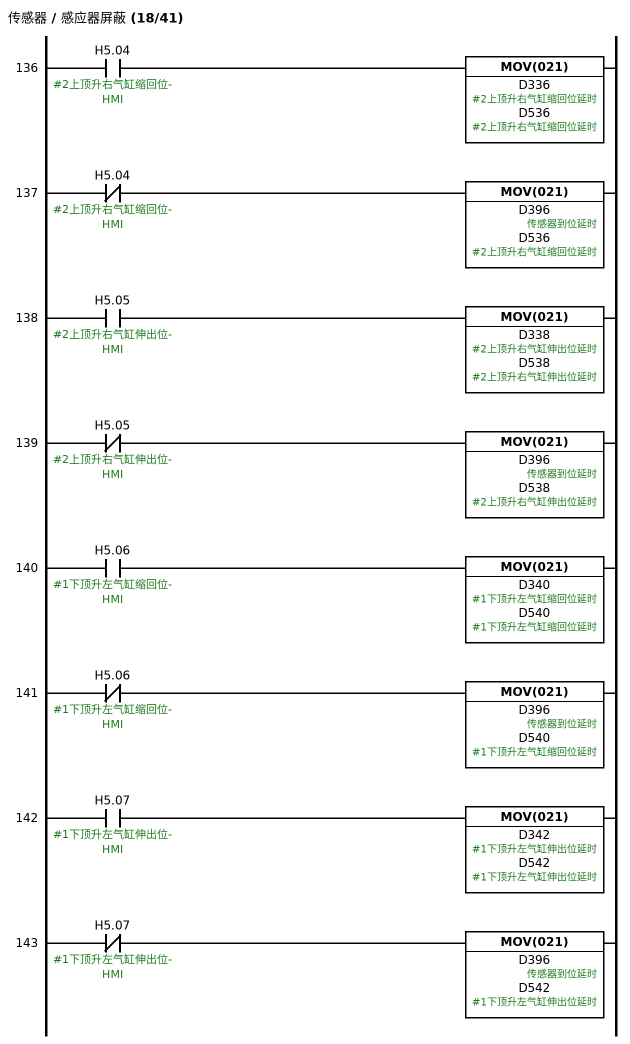
; rung 136
LD H5.04  ; #2上顶升右气缸缩回位-HMI
MOV(021) D336 D536  ; #2上顶升右气缸缩回位延时
; rung 137
LDNOT H5.04  ; #2上顶升右气缸缩回位-HMI
MOV(021) D396 D536  ; 传感器到位延时, #2上顶升右气缸缩回位延时
; rung 138
LD H5.05  ; #2上顶升右气缸伸出位-HMI
MOV(021) D338 D538  ; #2上顶升右气缸伸出位延时
; rung 139
LDNOT H5.05  ; #2上顶升右气缸伸出位-HMI
MOV(021) D396 D538  ; 传感器到位延时, #2上顶升右气缸伸出位延时
; rung 140
LD H5.06  ; #1下顶升左气缸缩回位-HMI
MOV(021) D340 D540  ; #1下顶升左气缸缩回位延时
; rung 141
LDNOT H5.06  ; #1下顶升左气缸缩回位-HMI
MOV(021) D396 D540  ; 传感器到位延时, #1下顶升左气缸缩回位延时
; rung 142
LD H5.07  ; #1下顶升左气缸伸出位-HMI
MOV(021) D342 D542  ; #1下顶升左气缸伸出位延时
; rung 143
LDNOT H5.07  ; #1下顶升左气缸伸出位-HMI
MOV(021) D396 D542  ; 传感器到位延时, #1下顶升左气缸伸出位延时

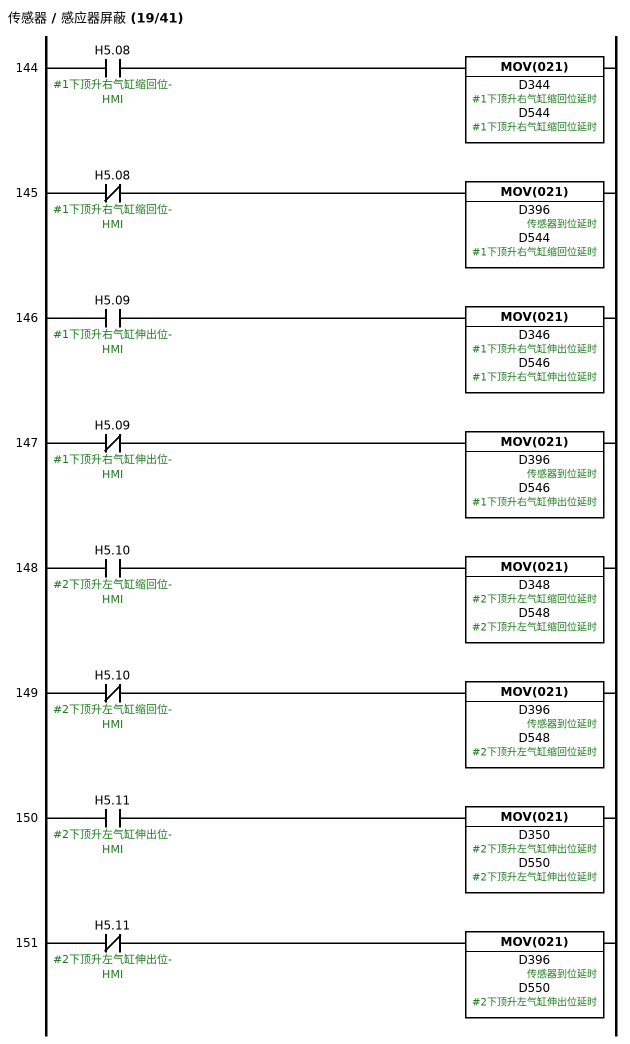
; rung 144
LD H5.08  ; #1下顶升右气缸缩回位-HMI
MOV(021) D344 D544  ; #1下顶升右气缸缩回位延时
; rung 145
LDNOT H5.08  ; #1下顶升右气缸缩回位-HMI
MOV(021) D396 D544  ; 传感器到位延时, #1下顶升右气缸缩回位延时
; rung 146
LD H5.09  ; #1下顶升右气缸伸出位-HMI
MOV(021) D346 D546  ; #1下顶升右气缸伸出位延时
; rung 147
LDNOT H5.09  ; #1下顶升右气缸伸出位-HMI
MOV(021) D396 D546  ; 传感器到位延时, #1下顶升右气缸伸出位延时
; rung 148
LD H5.10  ; #2下顶升左气缸缩回位-HMI
MOV(021) D348 D548  ; #2下顶升左气缸缩回位延时
; rung 149
LDNOT H5.10  ; #2下顶升左气缸缩回位-HMI
MOV(021) D396 D548  ; 传感器到位延时, #2下顶升左气缸缩回位延时
; rung 150
LD H5.11  ; #2下顶升左气缸伸出位-HMI
MOV(021) D350 D550  ; #2下顶升左气缸伸出位延时
; rung 151
LDNOT H5.11  ; #2下顶升左气缸伸出位-HMI
MOV(021) D396 D550  ; 传感器到位延时, #2下顶升左气缸伸出位延时

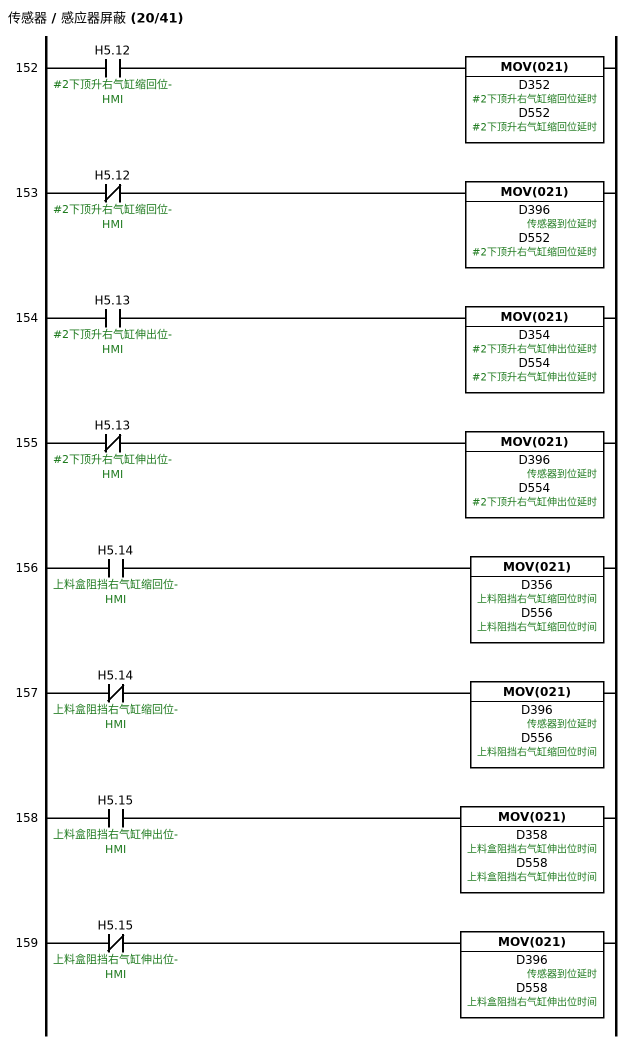
; rung 152
LD H5.12  ; #2下顶升右气缸缩回位-HMI
MOV(021) D352 D552  ; #2下顶升右气缸缩回位延时
; rung 153
LDNOT H5.12  ; #2下顶升右气缸缩回位-HMI
MOV(021) D396 D552  ; 传感器到位延时, #2下顶升右气缸缩回位延时
; rung 154
LD H5.13  ; #2下顶升右气缸伸出位-HMI
MOV(021) D354 D554  ; #2下顶升右气缸伸出位延时
; rung 155
LDNOT H5.13  ; #2下顶升右气缸伸出位-HMI
MOV(021) D396 D554  ; 传感器到位延时, #2下顶升右气缸伸出位延时
; rung 156
LD H5.14  ; 上料盒阻挡右气缸缩回位-HMI
MOV(021) D356 D556  ; 上料阻挡右气缸缩回位时间
; rung 157
LDNOT H5.14  ; 上料盒阻挡右气缸缩回位-HMI
MOV(021) D396 D556  ; 传感器到位延时, 上料阻挡右气缸缩回位时间
; rung 158
LD H5.15  ; 上料盒阻挡右气缸伸出位-HMI
MOV(021) D358 D558  ; 上料盒阻挡右气缸伸出位时间
; rung 159
LDNOT H5.15  ; 上料盒阻挡右气缸伸出位-HMI
MOV(021) D396 D558  ; 传感器到位延时, 上料盒阻挡右气缸伸出位时间

